TYPE ST_DALIBridgeInputEventParams :
STRUCT
	eventScheme 	: E_DALIEventScheme;
	addressInfo1 	: BYTE;
	addressInfo2 	: BYTE;
END_STRUCT
END_TYPE

(* stored: Version 1.1.0.1, ProductVersion 3.1.4024.10
   DUT ST_DALIBridgeInputEventParams: Id {bb798eac-7d3b-455f-8734-19a4f56fe226} *)
